PROGRAM MAIN
VAR
END_VAR

END_PROGRAM

(* stored: Version 1.1.0.1
   POU MAIN: Id {1218153c-87ee-43b2-a4f6-25aa934abf25} *)
